RoboDK station: a01274570_station.rdk

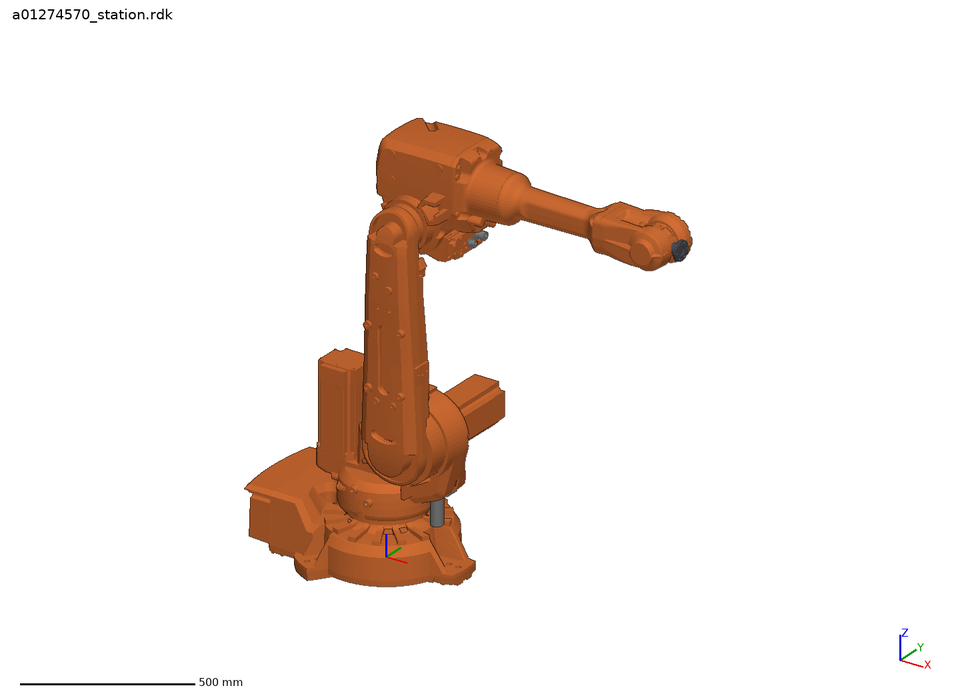
[picture v0: the station drawn from its stored meshes, robots at their saved joint values, targets as dots, program paths as lines]
Station a01274570_station (saved by RoboDK 5.5.0). Poses are relative to the parent item; angles as X-Y-Z fixed-axis rotations.
  - frame ABB IRB 2600-20/1.65 Base at (0, 0, 0) mm
    - robot ABB IRB 2600-20/1.65: 6 axes, payload 20 kg, reach 1650 mm, repeatability 0.04 mm, weight 272 kg
        modified DH rows (alpha deg, a mm, theta deg, d mm): 0, 0, 0, 445; -90, 150, -90, 0; 0, 700, 0, 0; -90, 115, 0, 795; 90, 0, 0, 0; -90, 0, 180, 85
        joint limits [-180, -95, -180, -400, -120, -400] to [180, 155, 75, 400, 120, 400]; home [0, 0, 0, 0, 0, 0]; saved at [0, 0, 0, 0, 0, 0]
